// TIA Portal V17 export
// export: Created 2025-04-22T12:08:41.9524589Z, ExportSetting WithDefaults, DisplayName Totally Integrated Automation Portal, DisplayVersion V17 Update 8, DisplayName TIA Portal Openness, DisplayVersion V17 Update 8, DisplayName TIA Portal Version Control Interface, DisplayVersion V17, DisplayName SINAMICS Startdrive Advanced, DisplayVersion V17 SP2, DisplayName SINAMICS Startdrive G110M, G120, G120C, G120D, G120P, G115D, DisplayVersion V17 SP2, DisplayName SINAMICS Startdrive G130, G150, S120, S150, SINAMICS MV, S210, DisplayVersion V17 SP2, DisplayName STEP 7 Professional, DisplayVersion V17 Update 8, DisplayName SINUMERIK ONE STEP 7 Toolbox, DisplayVersion V17 Update 12, DisplayName SINUMERIK 840D sl STEP 7 Toolbox, DisplayVersion V17 Update 12, DisplayName STEP 7 Safety, DisplayVersion V17 Update 6, DisplayName WinCC Advanced / Unified PC, DisplayVersion V17 Update 8
FUNCTION "FC20200_LASER_TRUMPF_READY" : Void   // FC20200, LAD
TITLE = FC20200 LASER TRUMPF READY
{ S7_Optimized_Access := 'TRUE' }
VERSION : 0.1
// stored: AutoNumber false, IsIECCheckEnabled false, SetENOAutomatically false, UDAEnableTagReadback false
   VAR_TEMP
      ret_val_1 : Int;
   END_VAR
BEGIN

REGION Network 1: LASER UNIT 01 INPUTS
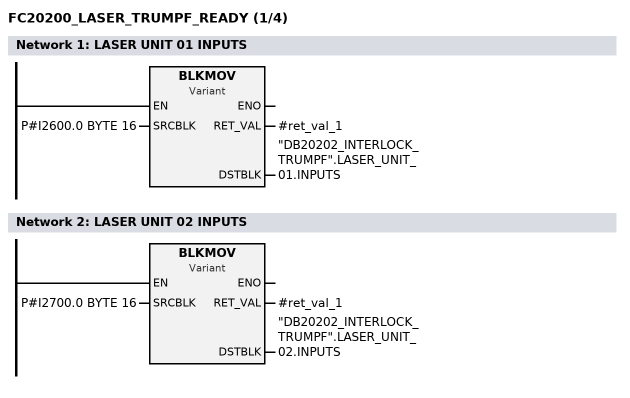
   RUNG wire#powerrail
      { S7_Templates := "blk_type := Variant" } BLKMOV(SRCBLK := P#I2600.0 BYTE 16, RET_VAL => #ret_val_1, DSTBLK => "DB20202_INTERLOCK_TRUMPF".LASER_UNIT_01.INPUTS)
   END_RUNG
   // the same network as SCL:
   #ret_val_1 := BLKMOV(SRCBLK := P#I2600.0 BYTE 16, DSTBLK => "DB20202_INTERLOCK_TRUMPF".LASER_UNIT_01.INPUTS);
END_REGION

REGION Network 2: LASER UNIT 02 INPUTS
   RUNG wire#powerrail
      { S7_Templates := "blk_type := Variant" } BLKMOV(SRCBLK := P#I2700.0 BYTE 16, RET_VAL => #ret_val_1, DSTBLK => "DB20202_INTERLOCK_TRUMPF".LASER_UNIT_02.INPUTS)
   END_RUNG
   // the same network as SCL:
   #ret_val_1 := BLKMOV(SRCBLK := P#I2700.0 BYTE 16, DSTBLK => "DB20202_INTERLOCK_TRUMPF".LASER_UNIT_02.INPUTS);
END_REGION

REGION Network 3: CALL LASER UNIT 01
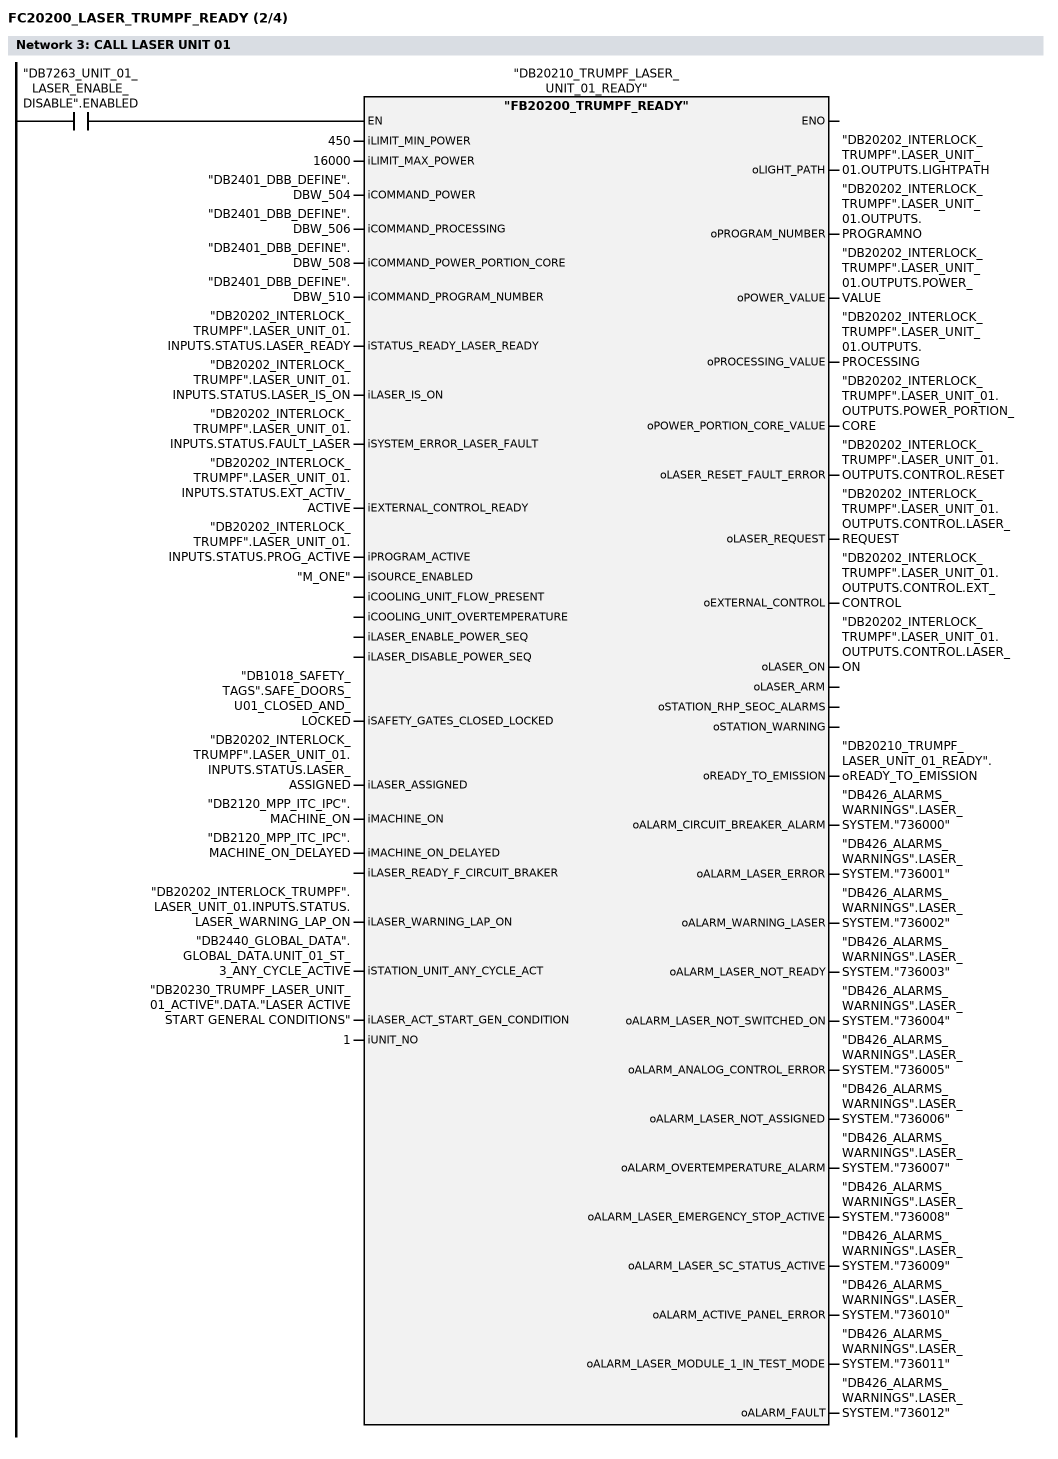
   RUNG wire#powerrail
      Contact( "DB7263_UNIT_01_LASER_ENABLE_DISABLE".ENABLED )
      "DB20210_TRUMPF_LASER_UNIT_01_READY"(iLIMIT_MIN_POWER := 450, iLIMIT_MAX_POWER := 16000, iCOMMAND_POWER := "DB2401_DBB_DEFINE".DBW_504, iCOMMAND_PROCESSING := "DB2401_DBB_DEFINE".DBW_506, iCOMMAND_POWER_PORTION_CORE := "DB2401_DBB_DEFINE".DBW_508, iCOMMAND_PROGRAM_NUMBER := "DB2401_DBB_DEFINE".DBW_510, iSTATUS_READY_LASER_READY := "DB20202_INTERLOCK_TRUMPF".LASER_UNIT_01.INPUTS.STATUS.LASER_READY, iLASER_IS_ON := "DB20202_INTERLOCK_TRUMPF".LASER_UNIT_01.INPUTS.STATUS.LASER_IS_ON, iSYSTEM_ERROR_LASER_FAULT := "DB20202_INTERLOCK_TRUMPF".LASER_UNIT_01.INPUTS.STATUS.FAULT_LASER, iEXTERNAL_CONTROL_READY := "DB20202_INTERLOCK_TRUMPF".LASER_UNIT_01.INPUTS.STATUS.EXT_ACTIV_ACTIVE, iPROGRAM_ACTIVE := "DB20202_INTERLOCK_TRUMPF".LASER_UNIT_01.INPUTS.STATUS.PROG_ACTIVE, iSOURCE_ENABLED := "M_ONE", iCOOLING_UNIT_FLOW_PRESENT :=, iCOOLING_UNIT_OVERTEMPERATURE :=, iLASER_ENABLE_POWER_SEQ :=, iLASER_DISABLE_POWER_SEQ :=, iSAFETY_GATES_CLOSED_LOCKED := "DB1018_SAFETY_TAGS".SAFE_DOORS_U01_CLOSED_AND_LOCKED, iLASER_ASSIGNED := "DB20202_INTERLOCK_TRUMPF".LASER_UNIT_01.INPUTS.STATUS.LASER_ASSIGNED, iMACHINE_ON := "DB2120_MPP_ITC_IPC".MACHINE_ON, iMACHINE_ON_DELAYED := "DB2120_MPP_ITC_IPC".MACHINE_ON_DELAYED, iLASER_READY_F_CIRCUIT_BRAKER :=, iLASER_WARNING_LAP_ON := "DB20202_INTERLOCK_TRUMPF".LASER_UNIT_01.INPUTS.STATUS.LASER_WARNING_LAP_ON, iSTATION_UNIT_ANY_CYCLE_ACT := "DB2440_GLOBAL_DATA".GLOBAL_DATA.UNIT_01_ST_3_ANY_CYCLE_ACTIVE, iLASER_ACT_START_GEN_CONDITION := "DB20230_TRUMPF_LASER_UNIT_01_ACTIVE".DATA."LASER ACTIVE START GENERAL CONDITIONS", iUNIT_NO := 1, oLIGHT_PATH => "DB20202_INTERLOCK_TRUMPF".LASER_UNIT_01.OUTPUTS.LIGHTPATH, oPROGRAM_NUMBER => "DB20202_INTERLOCK_TRUMPF".LASER_UNIT_01.OUTPUTS.PROGRAMNO, oPOWER_VALUE => "DB20202_INTERLOCK_TRUMPF".LASER_UNIT_01.OUTPUTS.POWER_VALUE, oPROCESSING_VALUE => "DB20202_INTERLOCK_TRUMPF".LASER_UNIT_01.OUTPUTS.PROCESSING, oPOWER_PORTION_CORE_VALUE => "DB20202_INTERLOCK_TRUMPF".LASER_UNIT_01.OUTPUTS.POWER_PORTION_CORE, oLASER_RESET_FAULT_ERROR => "DB20202_INTERLOCK_TRUMPF".LASER_UNIT_01.OUTPUTS.CONTROL.RESET, oLASER_REQUEST => "DB20202_INTERLOCK_TRUMPF".LASER_UNIT_01.OUTPUTS.CONTROL.LASER_REQUEST, oEXTERNAL_CONTROL => "DB20202_INTERLOCK_TRUMPF".LASER_UNIT_01.OUTPUTS.CONTROL.EXT_CONTROL, oLASER_ON => "DB20202_INTERLOCK_TRUMPF".LASER_UNIT_01.OUTPUTS.CONTROL.LASER_ON, oLASER_ARM =>, oSTATION_RHP_SEOC_ALARMS =>, oSTATION_WARNING =>, oREADY_TO_EMISSION => "DB20210_TRUMPF_LASER_UNIT_01_READY".oREADY_TO_EMISSION, oALARM_CIRCUIT_BREAKER_ALARM => "DB426_ALARMS_WARNINGS".LASER_SYSTEM."736000", oALARM_LASER_ERROR => "DB426_ALARMS_WARNINGS".LASER_SYSTEM."736001", oALARM_WARNING_LASER => "DB426_ALARMS_WARNINGS".LASER_SYSTEM."736002", oALARM_LASER_NOT_READY => "DB426_ALARMS_WARNINGS".LASER_SYSTEM."736003", oALARM_LASER_NOT_SWITCHED_ON => "DB426_ALARMS_WARNINGS".LASER_SYSTEM."736004", oALARM_ANALOG_CONTROL_ERROR => "DB426_ALARMS_WARNINGS".LASER_SYSTEM."736005", oALARM_LASER_NOT_ASSIGNED => "DB426_ALARMS_WARNINGS".LASER_SYSTEM."736006", oALARM_OVERTEMPERATURE_ALARM => "DB426_ALARMS_WARNINGS".LASER_SYSTEM."736007", oALARM_LASER_EMERGENCY_STOP_ACTIVE => "DB426_ALARMS_WARNINGS".LASER_SYSTEM."736008", oALARM_LASER_SC_STATUS_ACTIVE => "DB426_ALARMS_WARNINGS".LASER_SYSTEM."736009", oALARM_ACTIVE_PANEL_ERROR => "DB426_ALARMS_WARNINGS".LASER_SYSTEM."736010", oALARM_LASER_MODULE_1_IN_TEST_MODE => "DB426_ALARMS_WARNINGS".LASER_SYSTEM."736011", oALARM_FAULT => "DB426_ALARMS_WARNINGS".LASER_SYSTEM."736012")
   END_RUNG
   // the same network as SCL:
   IF "DB7263_UNIT_01_LASER_ENABLE_DISABLE".ENABLED THEN
       "DB20210_TRUMPF_LASER_UNIT_01_READY"(iLIMIT_MIN_POWER := 450,   // "FB20200_TRUMPF_READY"
                               iLIMIT_MAX_POWER := 16000,
                               iCOMMAND_POWER := "DB2401_DBB_DEFINE".DBW_504,
                               iCOMMAND_PROCESSING := "DB2401_DBB_DEFINE".DBW_506,
                               iCOMMAND_POWER_PORTION_CORE := "DB2401_DBB_DEFINE".DBW_508,
                               iCOMMAND_PROGRAM_NUMBER := "DB2401_DBB_DEFINE".DBW_510,
                               iSTATUS_READY_LASER_READY := "DB20202_INTERLOCK_TRUMPF".LASER_UNIT_01.INPUTS.STATUS.LASER_READY,
                               iLASER_IS_ON := "DB20202_INTERLOCK_TRUMPF".LASER_UNIT_01.INPUTS.STATUS.LASER_IS_ON,
                               iSYSTEM_ERROR_LASER_FAULT := "DB20202_INTERLOCK_TRUMPF".LASER_UNIT_01.INPUTS.STATUS.FAULT_LASER,
                               iEXTERNAL_CONTROL_READY := "DB20202_INTERLOCK_TRUMPF".LASER_UNIT_01.INPUTS.STATUS.EXT_ACTIV_ACTIVE,
                               iPROGRAM_ACTIVE := "DB20202_INTERLOCK_TRUMPF".LASER_UNIT_01.INPUTS.STATUS.PROG_ACTIVE,
                               iSOURCE_ENABLED := "M_ONE",
                               iSAFETY_GATES_CLOSED_LOCKED := "DB1018_SAFETY_TAGS".SAFE_DOORS_U01_CLOSED_AND_LOCKED,
                               iLASER_ASSIGNED := "DB20202_INTERLOCK_TRUMPF".LASER_UNIT_01.INPUTS.STATUS.LASER_ASSIGNED,
                               iMACHINE_ON := "DB2120_MPP_ITC_IPC".MACHINE_ON,
                               iMACHINE_ON_DELAYED := "DB2120_MPP_ITC_IPC".MACHINE_ON_DELAYED,
                               iLASER_WARNING_LAP_ON := "DB20202_INTERLOCK_TRUMPF".LASER_UNIT_01.INPUTS.STATUS.LASER_WARNING_LAP_ON,
                               iSTATION_UNIT_ANY_CYCLE_ACT := "DB2440_GLOBAL_DATA".GLOBAL_DATA.UNIT_01_ST_3_ANY_CYCLE_ACTIVE,
                               iLASER_ACT_START_GEN_CONDITION := "DB20230_TRUMPF_LASER_UNIT_01_ACTIVE".DATA."LASER ACTIVE START GENERAL CONDITIONS",
                               iUNIT_NO := 1,
                               oLIGHT_PATH => "DB20202_INTERLOCK_TRUMPF".LASER_UNIT_01.OUTPUTS.LIGHTPATH,
                               oPROGRAM_NUMBER => "DB20202_INTERLOCK_TRUMPF".LASER_UNIT_01.OUTPUTS.PROGRAMNO,
                               oPOWER_VALUE => "DB20202_INTERLOCK_TRUMPF".LASER_UNIT_01.OUTPUTS.POWER_VALUE,
                               oPROCESSING_VALUE => "DB20202_INTERLOCK_TRUMPF".LASER_UNIT_01.OUTPUTS.PROCESSING,
                               oPOWER_PORTION_CORE_VALUE => "DB20202_INTERLOCK_TRUMPF".LASER_UNIT_01.OUTPUTS.POWER_PORTION_CORE,
                               oLASER_RESET_FAULT_ERROR => "DB20202_INTERLOCK_TRUMPF".LASER_UNIT_01.OUTPUTS.CONTROL.RESET,
                               oLASER_REQUEST => "DB20202_INTERLOCK_TRUMPF".LASER_UNIT_01.OUTPUTS.CONTROL.LASER_REQUEST,
                               oEXTERNAL_CONTROL => "DB20202_INTERLOCK_TRUMPF".LASER_UNIT_01.OUTPUTS.CONTROL.EXT_CONTROL,
                               oLASER_ON => "DB20202_INTERLOCK_TRUMPF".LASER_UNIT_01.OUTPUTS.CONTROL.LASER_ON,
                               oREADY_TO_EMISSION => "DB20210_TRUMPF_LASER_UNIT_01_READY".oREADY_TO_EMISSION,
                               oALARM_CIRCUIT_BREAKER_ALARM => "DB426_ALARMS_WARNINGS".LASER_SYSTEM."736000",
                               oALARM_LASER_ERROR => "DB426_ALARMS_WARNINGS".LASER_SYSTEM."736001",
                               oALARM_WARNING_LASER => "DB426_ALARMS_WARNINGS".LASER_SYSTEM."736002",
                               oALARM_LASER_NOT_READY => "DB426_ALARMS_WARNINGS".LASER_SYSTEM."736003",
                               oALARM_LASER_NOT_SWITCHED_ON => "DB426_ALARMS_WARNINGS".LASER_SYSTEM."736004",
                               oALARM_ANALOG_CONTROL_ERROR => "DB426_ALARMS_WARNINGS".LASER_SYSTEM."736005",
                               oALARM_LASER_NOT_ASSIGNED => "DB426_ALARMS_WARNINGS".LASER_SYSTEM."736006",
                               oALARM_OVERTEMPERATURE_ALARM => "DB426_ALARMS_WARNINGS".LASER_SYSTEM."736007",
                               oALARM_LASER_EMERGENCY_STOP_ACTIVE => "DB426_ALARMS_WARNINGS".LASER_SYSTEM."736008",
                               oALARM_LASER_SC_STATUS_ACTIVE => "DB426_ALARMS_WARNINGS".LASER_SYSTEM."736009",
                               oALARM_ACTIVE_PANEL_ERROR => "DB426_ALARMS_WARNINGS".LASER_SYSTEM."736010",
                               oALARM_LASER_MODULE_1_IN_TEST_MODE => "DB426_ALARMS_WARNINGS".LASER_SYSTEM."736011",
                               oALARM_FAULT => "DB426_ALARMS_WARNINGS".LASER_SYSTEM."736012");
   END_IF;
END_REGION

REGION Network 4: CALL LASER UNIT 02
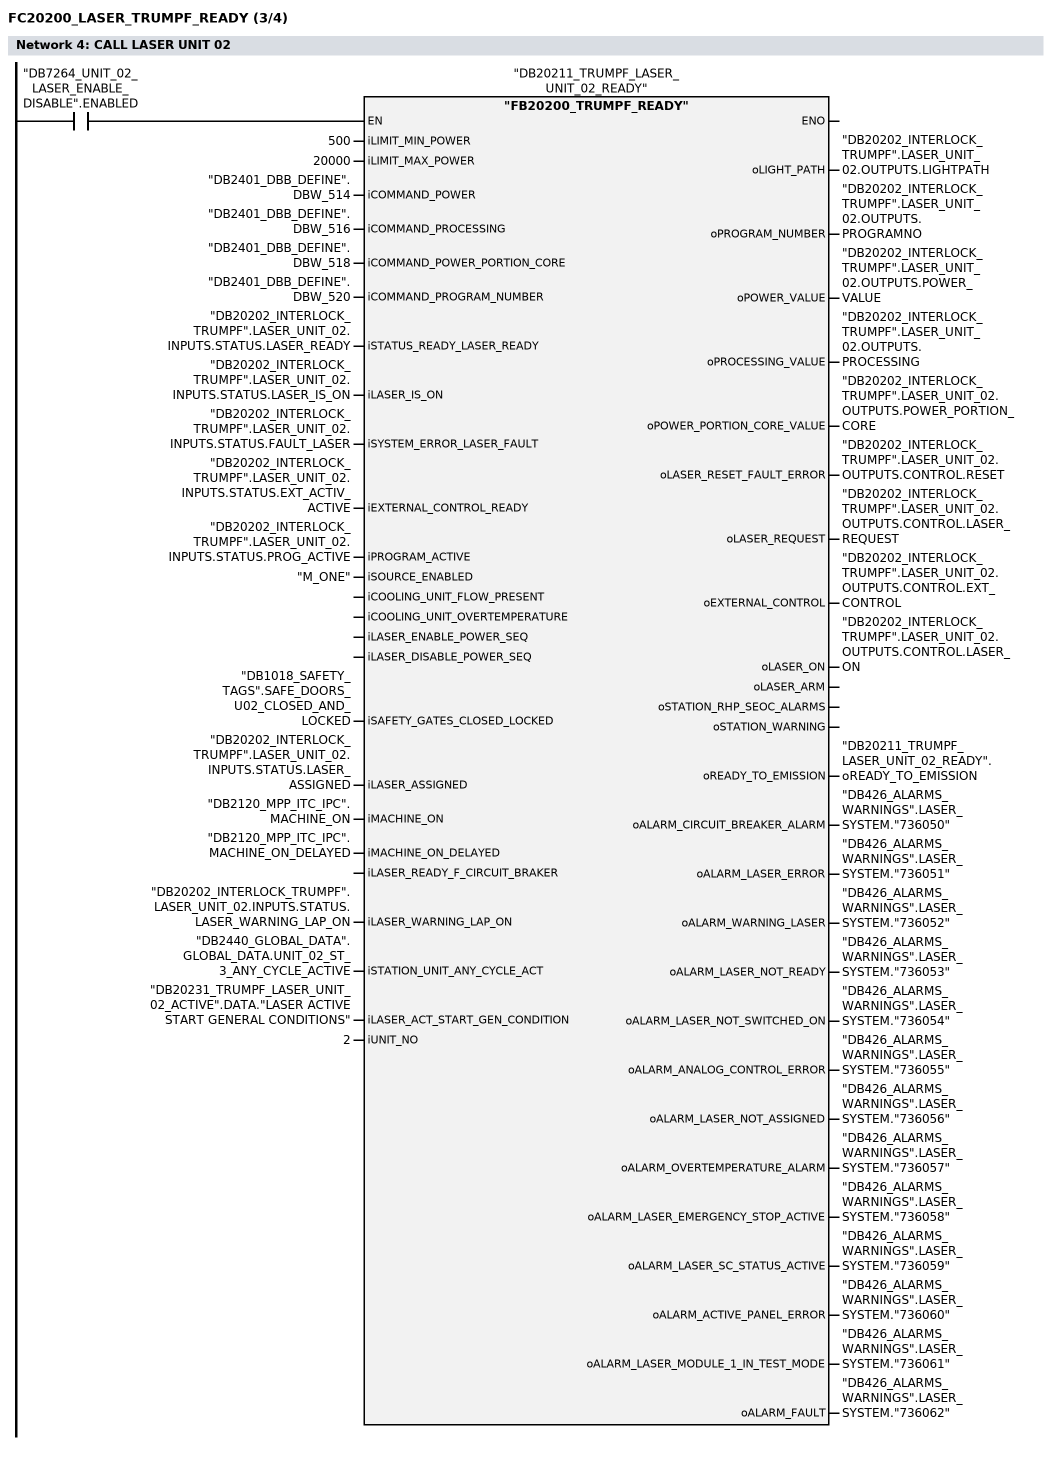
   RUNG wire#powerrail
      Contact( "DB7264_UNIT_02_LASER_ENABLE_DISABLE".ENABLED )
      "DB20211_TRUMPF_LASER_UNIT_02_READY"(iLIMIT_MIN_POWER := 500, iLIMIT_MAX_POWER := 20000, iCOMMAND_POWER := "DB2401_DBB_DEFINE".DBW_514, iCOMMAND_PROCESSING := "DB2401_DBB_DEFINE".DBW_516, iCOMMAND_POWER_PORTION_CORE := "DB2401_DBB_DEFINE".DBW_518, iCOMMAND_PROGRAM_NUMBER := "DB2401_DBB_DEFINE".DBW_520, iSTATUS_READY_LASER_READY := "DB20202_INTERLOCK_TRUMPF".LASER_UNIT_02.INPUTS.STATUS.LASER_READY, iLASER_IS_ON := "DB20202_INTERLOCK_TRUMPF".LASER_UNIT_02.INPUTS.STATUS.LASER_IS_ON, iSYSTEM_ERROR_LASER_FAULT := "DB20202_INTERLOCK_TRUMPF".LASER_UNIT_02.INPUTS.STATUS.FAULT_LASER, iEXTERNAL_CONTROL_READY := "DB20202_INTERLOCK_TRUMPF".LASER_UNIT_02.INPUTS.STATUS.EXT_ACTIV_ACTIVE, iPROGRAM_ACTIVE := "DB20202_INTERLOCK_TRUMPF".LASER_UNIT_02.INPUTS.STATUS.PROG_ACTIVE, iSOURCE_ENABLED := "M_ONE", iCOOLING_UNIT_FLOW_PRESENT :=, iCOOLING_UNIT_OVERTEMPERATURE :=, iLASER_ENABLE_POWER_SEQ :=, iLASER_DISABLE_POWER_SEQ :=, iSAFETY_GATES_CLOSED_LOCKED := "DB1018_SAFETY_TAGS".SAFE_DOORS_U02_CLOSED_AND_LOCKED, iLASER_ASSIGNED := "DB20202_INTERLOCK_TRUMPF".LASER_UNIT_02.INPUTS.STATUS.LASER_ASSIGNED, iMACHINE_ON := "DB2120_MPP_ITC_IPC".MACHINE_ON, iMACHINE_ON_DELAYED := "DB2120_MPP_ITC_IPC".MACHINE_ON_DELAYED, iLASER_READY_F_CIRCUIT_BRAKER :=, iLASER_WARNING_LAP_ON := "DB20202_INTERLOCK_TRUMPF".LASER_UNIT_02.INPUTS.STATUS.LASER_WARNING_LAP_ON, iSTATION_UNIT_ANY_CYCLE_ACT := "DB2440_GLOBAL_DATA".GLOBAL_DATA.UNIT_02_ST_3_ANY_CYCLE_ACTIVE, iLASER_ACT_START_GEN_CONDITION := "DB20231_TRUMPF_LASER_UNIT_02_ACTIVE".DATA."LASER ACTIVE START GENERAL CONDITIONS", iUNIT_NO := 2, oLIGHT_PATH => "DB20202_INTERLOCK_TRUMPF".LASER_UNIT_02.OUTPUTS.LIGHTPATH, oPROGRAM_NUMBER => "DB20202_INTERLOCK_TRUMPF".LASER_UNIT_02.OUTPUTS.PROGRAMNO, oPOWER_VALUE => "DB20202_INTERLOCK_TRUMPF".LASER_UNIT_02.OUTPUTS.POWER_VALUE, oPROCESSING_VALUE => "DB20202_INTERLOCK_TRUMPF".LASER_UNIT_02.OUTPUTS.PROCESSING, oPOWER_PORTION_CORE_VALUE => "DB20202_INTERLOCK_TRUMPF".LASER_UNIT_02.OUTPUTS.POWER_PORTION_CORE, oLASER_RESET_FAULT_ERROR => "DB20202_INTERLOCK_TRUMPF".LASER_UNIT_02.OUTPUTS.CONTROL.RESET, oLASER_REQUEST => "DB20202_INTERLOCK_TRUMPF".LASER_UNIT_02.OUTPUTS.CONTROL.LASER_REQUEST, oEXTERNAL_CONTROL => "DB20202_INTERLOCK_TRUMPF".LASER_UNIT_02.OUTPUTS.CONTROL.EXT_CONTROL, oLASER_ON => "DB20202_INTERLOCK_TRUMPF".LASER_UNIT_02.OUTPUTS.CONTROL.LASER_ON, oLASER_ARM =>, oSTATION_RHP_SEOC_ALARMS =>, oSTATION_WARNING =>, oREADY_TO_EMISSION => "DB20211_TRUMPF_LASER_UNIT_02_READY".oREADY_TO_EMISSION, oALARM_CIRCUIT_BREAKER_ALARM => "DB426_ALARMS_WARNINGS".LASER_SYSTEM."736050", oALARM_LASER_ERROR => "DB426_ALARMS_WARNINGS".LASER_SYSTEM."736051", oALARM_WARNING_LASER => "DB426_ALARMS_WARNINGS".LASER_SYSTEM."736052", oALARM_LASER_NOT_READY => "DB426_ALARMS_WARNINGS".LASER_SYSTEM."736053", oALARM_LASER_NOT_SWITCHED_ON => "DB426_ALARMS_WARNINGS".LASER_SYSTEM."736054", oALARM_ANALOG_CONTROL_ERROR => "DB426_ALARMS_WARNINGS".LASER_SYSTEM."736055", oALARM_LASER_NOT_ASSIGNED => "DB426_ALARMS_WARNINGS".LASER_SYSTEM."736056", oALARM_OVERTEMPERATURE_ALARM => "DB426_ALARMS_WARNINGS".LASER_SYSTEM."736057", oALARM_LASER_EMERGENCY_STOP_ACTIVE => "DB426_ALARMS_WARNINGS".LASER_SYSTEM."736058", oALARM_LASER_SC_STATUS_ACTIVE => "DB426_ALARMS_WARNINGS".LASER_SYSTEM."736059", oALARM_ACTIVE_PANEL_ERROR => "DB426_ALARMS_WARNINGS".LASER_SYSTEM."736060", oALARM_LASER_MODULE_1_IN_TEST_MODE => "DB426_ALARMS_WARNINGS".LASER_SYSTEM."736061", oALARM_FAULT => "DB426_ALARMS_WARNINGS".LASER_SYSTEM."736062")
   END_RUNG
   // the same network as SCL:
   IF "DB7264_UNIT_02_LASER_ENABLE_DISABLE".ENABLED THEN
       "DB20211_TRUMPF_LASER_UNIT_02_READY"(iLIMIT_MIN_POWER := 500,   // "FB20200_TRUMPF_READY"
                               iLIMIT_MAX_POWER := 20000,
                               iCOMMAND_POWER := "DB2401_DBB_DEFINE".DBW_514,
                               iCOMMAND_PROCESSING := "DB2401_DBB_DEFINE".DBW_516,
                               iCOMMAND_POWER_PORTION_CORE := "DB2401_DBB_DEFINE".DBW_518,
                               iCOMMAND_PROGRAM_NUMBER := "DB2401_DBB_DEFINE".DBW_520,
                               iSTATUS_READY_LASER_READY := "DB20202_INTERLOCK_TRUMPF".LASER_UNIT_02.INPUTS.STATUS.LASER_READY,
                               iLASER_IS_ON := "DB20202_INTERLOCK_TRUMPF".LASER_UNIT_02.INPUTS.STATUS.LASER_IS_ON,
                               iSYSTEM_ERROR_LASER_FAULT := "DB20202_INTERLOCK_TRUMPF".LASER_UNIT_02.INPUTS.STATUS.FAULT_LASER,
                               iEXTERNAL_CONTROL_READY := "DB20202_INTERLOCK_TRUMPF".LASER_UNIT_02.INPUTS.STATUS.EXT_ACTIV_ACTIVE,
                               iPROGRAM_ACTIVE := "DB20202_INTERLOCK_TRUMPF".LASER_UNIT_02.INPUTS.STATUS.PROG_ACTIVE,
                               iSOURCE_ENABLED := "M_ONE",
                               iSAFETY_GATES_CLOSED_LOCKED := "DB1018_SAFETY_TAGS".SAFE_DOORS_U02_CLOSED_AND_LOCKED,
                               iLASER_ASSIGNED := "DB20202_INTERLOCK_TRUMPF".LASER_UNIT_02.INPUTS.STATUS.LASER_ASSIGNED,
                               iMACHINE_ON := "DB2120_MPP_ITC_IPC".MACHINE_ON,
                               iMACHINE_ON_DELAYED := "DB2120_MPP_ITC_IPC".MACHINE_ON_DELAYED,
                               iLASER_WARNING_LAP_ON := "DB20202_INTERLOCK_TRUMPF".LASER_UNIT_02.INPUTS.STATUS.LASER_WARNING_LAP_ON,
                               iSTATION_UNIT_ANY_CYCLE_ACT := "DB2440_GLOBAL_DATA".GLOBAL_DATA.UNIT_02_ST_3_ANY_CYCLE_ACTIVE,
                               iLASER_ACT_START_GEN_CONDITION := "DB20231_TRUMPF_LASER_UNIT_02_ACTIVE".DATA."LASER ACTIVE START GENERAL CONDITIONS",
                               iUNIT_NO := 2,
                               oLIGHT_PATH => "DB20202_INTERLOCK_TRUMPF".LASER_UNIT_02.OUTPUTS.LIGHTPATH,
                               oPROGRAM_NUMBER => "DB20202_INTERLOCK_TRUMPF".LASER_UNIT_02.OUTPUTS.PROGRAMNO,
                               oPOWER_VALUE => "DB20202_INTERLOCK_TRUMPF".LASER_UNIT_02.OUTPUTS.POWER_VALUE,
                               oPROCESSING_VALUE => "DB20202_INTERLOCK_TRUMPF".LASER_UNIT_02.OUTPUTS.PROCESSING,
                               oPOWER_PORTION_CORE_VALUE => "DB20202_INTERLOCK_TRUMPF".LASER_UNIT_02.OUTPUTS.POWER_PORTION_CORE,
                               oLASER_RESET_FAULT_ERROR => "DB20202_INTERLOCK_TRUMPF".LASER_UNIT_02.OUTPUTS.CONTROL.RESET,
                               oLASER_REQUEST => "DB20202_INTERLOCK_TRUMPF".LASER_UNIT_02.OUTPUTS.CONTROL.LASER_REQUEST,
                               oEXTERNAL_CONTROL => "DB20202_INTERLOCK_TRUMPF".LASER_UNIT_02.OUTPUTS.CONTROL.EXT_CONTROL,
                               oLASER_ON => "DB20202_INTERLOCK_TRUMPF".LASER_UNIT_02.OUTPUTS.CONTROL.LASER_ON,
                               oREADY_TO_EMISSION => "DB20211_TRUMPF_LASER_UNIT_02_READY".oREADY_TO_EMISSION,
                               oALARM_CIRCUIT_BREAKER_ALARM => "DB426_ALARMS_WARNINGS".LASER_SYSTEM."736050",
                               oALARM_LASER_ERROR => "DB426_ALARMS_WARNINGS".LASER_SYSTEM."736051",
                               oALARM_WARNING_LASER => "DB426_ALARMS_WARNINGS".LASER_SYSTEM."736052",
                               oALARM_LASER_NOT_READY => "DB426_ALARMS_WARNINGS".LASER_SYSTEM."736053",
                               oALARM_LASER_NOT_SWITCHED_ON => "DB426_ALARMS_WARNINGS".LASER_SYSTEM."736054",
                               oALARM_ANALOG_CONTROL_ERROR => "DB426_ALARMS_WARNINGS".LASER_SYSTEM."736055",
                               oALARM_LASER_NOT_ASSIGNED => "DB426_ALARMS_WARNINGS".LASER_SYSTEM."736056",
                               oALARM_OVERTEMPERATURE_ALARM => "DB426_ALARMS_WARNINGS".LASER_SYSTEM."736057",
                               oALARM_LASER_EMERGENCY_STOP_ACTIVE => "DB426_ALARMS_WARNINGS".LASER_SYSTEM."736058",
                               oALARM_LASER_SC_STATUS_ACTIVE => "DB426_ALARMS_WARNINGS".LASER_SYSTEM."736059",
                               oALARM_ACTIVE_PANEL_ERROR => "DB426_ALARMS_WARNINGS".LASER_SYSTEM."736060",
                               oALARM_LASER_MODULE_1_IN_TEST_MODE => "DB426_ALARMS_WARNINGS".LASER_SYSTEM."736061",
                               oALARM_FAULT => "DB426_ALARMS_WARNINGS".LASER_SYSTEM."736062");
   END_IF;
END_REGION

REGION Network 5: ALL LASER READY
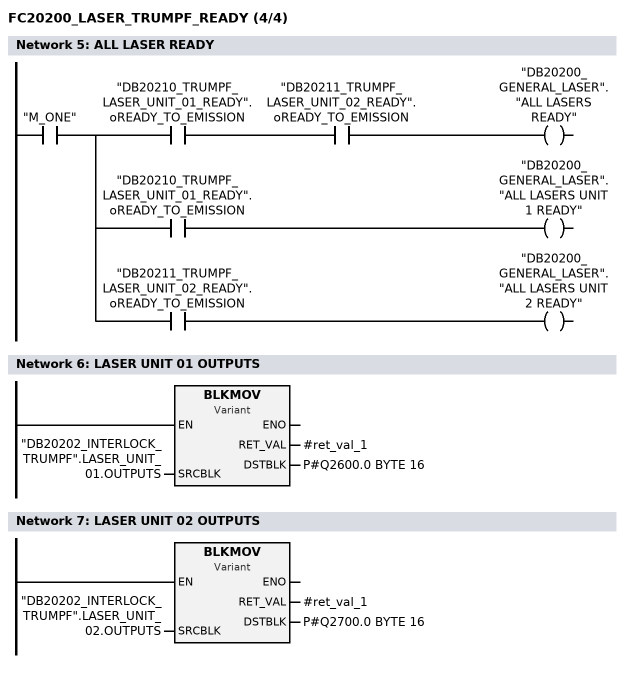
   RUNG wire#powerrail
      Contact( "M_ONE" )
      wire#w1
      Contact( "DB20210_TRUMPF_LASER_UNIT_01_READY".oREADY_TO_EMISSION )
      Contact( "DB20211_TRUMPF_LASER_UNIT_02_READY".oREADY_TO_EMISSION )
      Coil( "DB20200_GENERAL_LASER"."ALL LASERS READY" )
   END_RUNG
   RUNG wire#w1
      Contact( "DB20210_TRUMPF_LASER_UNIT_01_READY".oREADY_TO_EMISSION )
      Coil( "DB20200_GENERAL_LASER"."ALL LASERS UNIT 1 READY" )
   END_RUNG
   RUNG wire#w1
      Contact( "DB20211_TRUMPF_LASER_UNIT_02_READY".oREADY_TO_EMISSION )
      Coil( "DB20200_GENERAL_LASER"."ALL LASERS UNIT 2 READY" )
   END_RUNG
   // the same network as SCL:
   "DB20200_GENERAL_LASER"."ALL LASERS READY" := "M_ONE" AND "DB20210_TRUMPF_LASER_UNIT_01_READY".oREADY_TO_EMISSION AND "DB20211_TRUMPF_LASER_UNIT_02_READY".oREADY_TO_EMISSION;
   "DB20200_GENERAL_LASER"."ALL LASERS UNIT 1 READY" := "M_ONE" AND "DB20210_TRUMPF_LASER_UNIT_01_READY".oREADY_TO_EMISSION;
   "DB20200_GENERAL_LASER"."ALL LASERS UNIT 2 READY" := "M_ONE" AND "DB20211_TRUMPF_LASER_UNIT_02_READY".oREADY_TO_EMISSION;
END_REGION

REGION Network 6: LASER UNIT 01 OUTPUTS
   RUNG wire#powerrail
      { S7_Templates := "blk_type := Variant" } BLKMOV(SRCBLK := "DB20202_INTERLOCK_TRUMPF".LASER_UNIT_01.OUTPUTS, RET_VAL => #ret_val_1, DSTBLK => P#Q2600.0 BYTE 16)
   END_RUNG
   // the same network as SCL:
   #ret_val_1 := BLKMOV(SRCBLK := "DB20202_INTERLOCK_TRUMPF".LASER_UNIT_01.OUTPUTS, DSTBLK => P#Q2600.0 BYTE 16);
END_REGION

REGION Network 7: LASER UNIT 02 OUTPUTS
   RUNG wire#powerrail
      { S7_Templates := "blk_type := Variant" } BLKMOV(SRCBLK := "DB20202_INTERLOCK_TRUMPF".LASER_UNIT_02.OUTPUTS, RET_VAL => #ret_val_1, DSTBLK => P#Q2700.0 BYTE 16)
   END_RUNG
   // the same network as SCL:
   #ret_val_1 := BLKMOV(SRCBLK := "DB20202_INTERLOCK_TRUMPF".LASER_UNIT_02.OUTPUTS, DSTBLK => P#Q2700.0 BYTE 16);
END_REGION
END_FUNCTION
